FUNCTION_BLOCK FB_MoverList
VAR_OUTPUT	
	List									: ARRAY[0..MAX_MOVERS] OF INT; //starts from 0, element zero is the number in the list 
END_VAR
VAR
	i: INT;
END_VAR

// Adding and removing stuff to a list can be a difficult as such a block has 
// been built with methods to add/remove from a list. 
// list acts like a FIFO, the list is filled from the back and emptied from the front.

METHOD M_AddToList
VAR_INPUT
	IDToAdd: INT;
END_VAR
// Movers are handled in a FIFO manner new movers are added to the end of the list 
List[0] 					:= List[0] +1; //List[0] holds the number of movers in the list 
List[List[0]] 				:= IDToAdd; //whern there is 1 in the list, List[0] = 1 and LIst[1] = IDToAdd
END_METHOD

METHOD M_ClearList
MEMSET(destAddr:=ADR(List),fillByte:=0,n:=SIZEOF(List));
END_METHOD

METHOD M_CopyList
VAR_INPUT
	ListToCopy: ARRAY[0..MAX_MOVERS] OF INT;
END_VAR
// method to copy a complete list, don't allow an extrnal copy unless its with a method
List := ListToCopy;
END_METHOD

METHOD M_GetFirstInList : INT
M_GetFirstInList := List[1];
END_METHOD

METHOD M_RecycleDown : BOOL
VAR
	iTemp: INT;
END_VAR
iTemp							:= List[MAX_MOVERS];
MEMCPY(ADR(List[2]),ADR(List[1]),SIZEOF(List)-SIZEOF(List[1])*2);
List[1]							:=iTemp;
M_RecycleDown					:= TRUE;
END_METHOD

METHOD M_RemoveFromList : INT
VAR
	I: INT;
END_VAR
//If there is something in the list, get the first element 
IF List[0] >= 1 THEN 
	M_RemoveFromList := List[1]; //List [1] is the first in the list, list[0] contains the number of items in the list  
	MEMCPY(ADR(List[1]),ADR(List[2]),SIZEOF(List)- 2 * SIZEOF(List[1])); //start at address 2 and copy the size of the list minus elements 0 and 1 
	List[MAX_MOVERS] := -1; //the last item in the list is now -1 
	List[0] := List[0]-1; // there is now one less item in the list 
ELSE //there was nothing in the list, return an invalid mover number 
	M_RemoveFromList := -1;// return an invalid mover 
END_IF
END_METHOD

METHOD M_RemoveLastFromList : int
VAR_INPUT
END_VAR
IF List[0] >= 1 THEN 
	M_RemoveLastFromList := List[ List[0]]; //List [1] is the first in the list, list[0] contains the number of items in the list  
	List[ List[0]]:=0;
	List[0]:=List[0]-1;
ELSE //there was nothing in the list, return an invalid mover number 
	M_RemoveLastFromList := -1;// return an invalid mover 
END_IF
END_METHOD

METHOD M_ReverseList : BOOL
VAR
	TempList: ARRAY[0..MAX_MOVERS] OF INT;
END_VAR
 
TempList:=List;
FOR i:=1 TO TempList[0] DO
	List[i]						:=TempList[TempList[0]+1-i];
END_FOR
M_ReverseList					:= TRUE;
END_METHOD

PROPERTY P_NumInList : INT
GET
P_NumInList:= List[0];
END_GET
END_PROPERTY

END_FUNCTION_BLOCK

(* stored: Version 1.1.0.1, ProductVersion 3.1.4024.12
   POU FB_MoverList: Id {a2667dab-69b3-4175-8c22-d7e1cc85801c}, SpecialFunc None
   Method M_AddToList: Id {5b9e86a5-a158-427c-97ec-d124d4eb6f67}
   Method M_ClearList: Id {347f8aed-0cdc-4834-a469-64c7c83ac020}
   Method M_CopyList: Id {23b7a85d-6afb-44c8-8b8c-26e12ba0cac3}
   Method M_GetFirstInList: Id {6f4ba9d2-1c2a-466d-838d-e3fceedf2714}
   Method M_RecycleDown: Id {d1614f47-eee1-4fa3-aba0-795ae06e52cf}
   Method M_RemoveFromList: Id {43c80c11-fff1-4b41-8cf6-b01765332bc3}
   Method M_RemoveLastFromList: Id {1c0be62f-280e-4c15-a34f-d0f364bee233}
   Method M_ReverseList: Id {62fde437-6f30-4513-b4a1-f60f6afc62c2}
   Property P_NumInList: Id {a7ec8362-0726-40db-a159-b3a05573917b}
   Get Get: Id {4e7b17d0-eee7-47a5-a720-101411499c9e} *)
